// TIA Portal V18 export
TYPE "UDT_Recipe_PressCurve"
// NOTE: UDT_Recipe_PressCurve and UDT_Recipe_ATEQ are assumed to exist from original project files.
//  =================================================================================
//  MAIN RECIPE UDT - FINAL VERSION
//  =================================================================================
   STRUCT
      StartPos_UL : Real;
      StartPos_LL : Real;
      StartForce_UL : Real;
      StartForce_LL : Real;
      MiddlePos_UL : Real;
      MiddlePos_LL : Real;
      MiddleForce_UL : Real;
      MiddleForce_LL : Real;
      FinalPos_UL : Real;
      FinalPos_LL : Real;
      FinalForce_UL : Real;
      FinalForce_LL : Real;
      ProgramNum : Int;
   END_STRUCT;
END_TYPE
